FUNCTION F_selu : lreal
VAR_INPUT
	x : LREAL;
END_VAR
VAR
	scale : LREAL := 1.05070098;
	alpha : LREAL := 1.67326324;
END_VAR

IF x > 0 THEN
	F_selu := scale * x;
ELSIF x < -10E6 THEN
	F_selu := - scale * alpha;
ELSE
	F_selu := scale * alpha * (exp(x) - 1);
END_IF

END_FUNCTION

(* stored: Version 1.1.0.1, ProductVersion 3.1.4024.12
   POU F_selu: Id {5f7120d9-0147-4b07-8c1a-9793deff443a}, SpecialFunc None *)
